FUNCTION_BLOCK FB_Tools
VAR_INPUT
END_VAR
VAR_OUTPUT
END_VAR
VAR
END_VAR

END_FUNCTION_BLOCK

(* stored: Version 1.1.0.1
   POU FB_Tools: Id {3b15b15d-aac5-4ba5-b61a-9a131ed1d0dc}, SpecialFunc None *)
